// Mitsubishi GX Works2 project: plc+hmi1   PLC: Q03UDV

PROGRAM MAIN
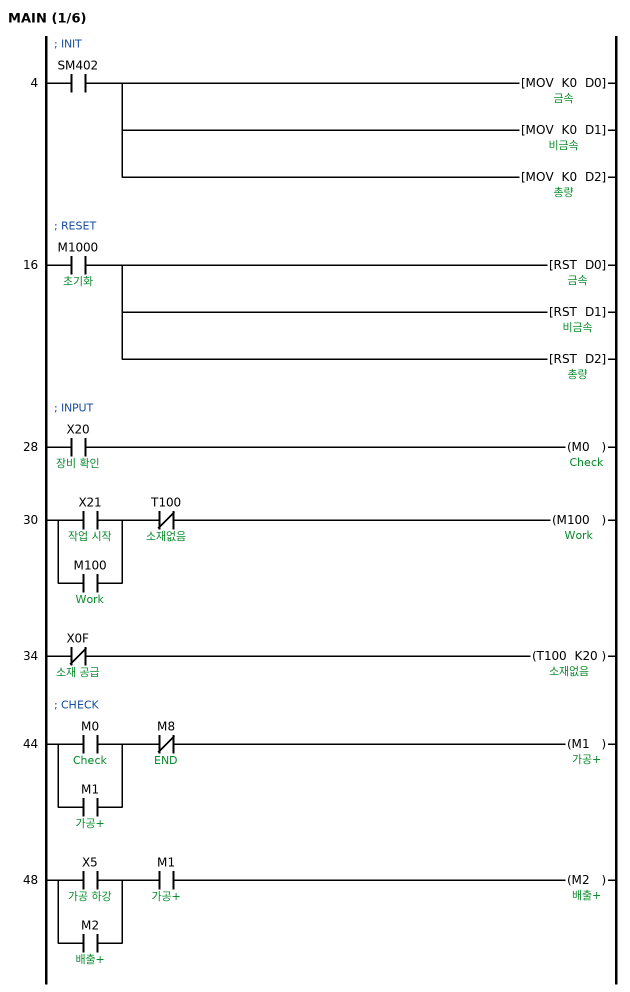
; INIT
4     LD      SM402
      MOV     K0 D0  ; 금속
      MOV     K0 D1  ; 비금속
      MOV     K0 D2  ; 총량
; RESET
16    LD      M1000  ; 초기화
      RST     D0  ; 금속
      RST     D1  ; 비금속
      RST     D2  ; 총량
; INPUT
28    LD      X20  ; 장비 확인
      OUT     M0  ; Check
30    LD      X21  ; 작업 시작
      OR      M100  ; Work
      ANI     T100  ; 소재없음
      OUT     M100  ; Work
34    LDI     X0F  ; 소재 공급
      OUT     T100 K20  ; 소재없음
; CHECK
44    LD      M0  ; Check
      OR      M1  ; 가공+
      ANI     M8  ; END
      OUT     M1  ; 가공+
48    LD      X5  ; 가공 하강
      OR      M2  ; 배출+
      AND     M1  ; 가공+
      OUT     M2  ; 배출+
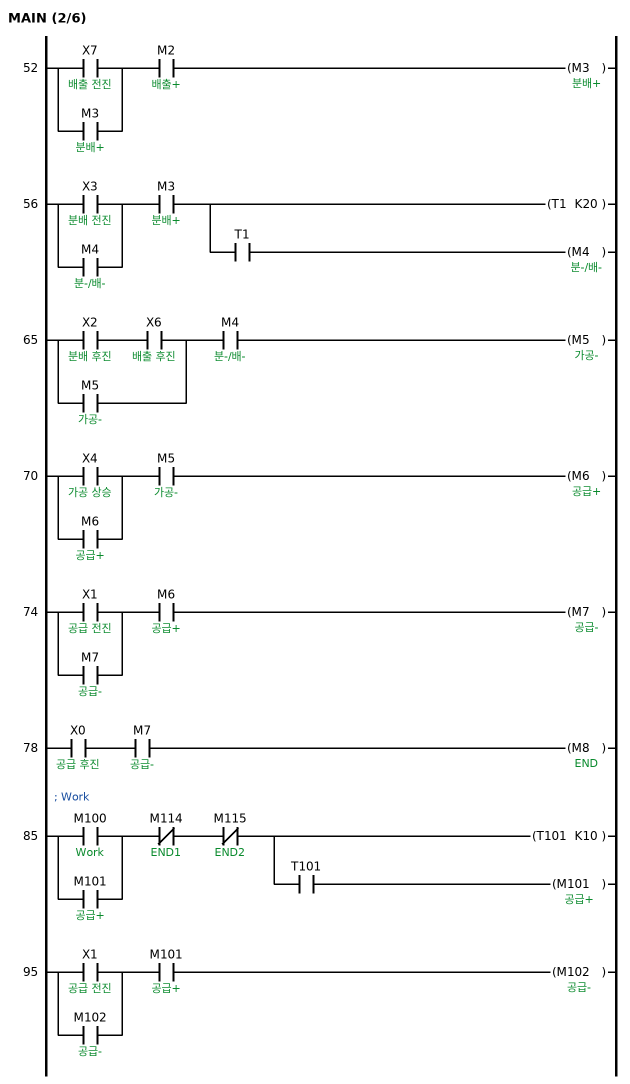
52    LD      X7  ; 배출 전진
      OR      M3  ; 분배+
      AND     M2  ; 배출+
      OUT     M3  ; 분배+
56    LD      X3  ; 분배 전진
      OR      M4  ; 분-/배-
      AND     M3  ; 분배+
      OUT     T1 K20
      AND     T1
      OUT     M4  ; 분-/배-
65    LD      X2  ; 분배 후진
      AND     X6  ; 배출 후진
      OR      M5  ; 가공-
      AND     M4  ; 분-/배-
      OUT     M5  ; 가공-
70    LD      X4  ; 가공 상승
      OR      M6  ; 공급+
      AND     M5  ; 가공-
      OUT     M6  ; 공급+
74    LD      X1  ; 공급 전진
      OR      M7  ; 공급-
      AND     M6  ; 공급+
      OUT     M7  ; 공급-
78    LD      X0  ; 공급 후진
      AND     M7  ; 공급-
      OUT     M8  ; END
; Work
85    LD      M100  ; Work
      OR      M101  ; 공급+
      ANI     M114  ; END1
      ANI     M115  ; END2
      OUT     T101 K10
      AND     T101
      OUT     M101  ; 공급+
95    LD      X1  ; 공급 전진
      OR      M102  ; 공급-
      AND     M101  ; 공급+
      OUT     M102  ; 공급-
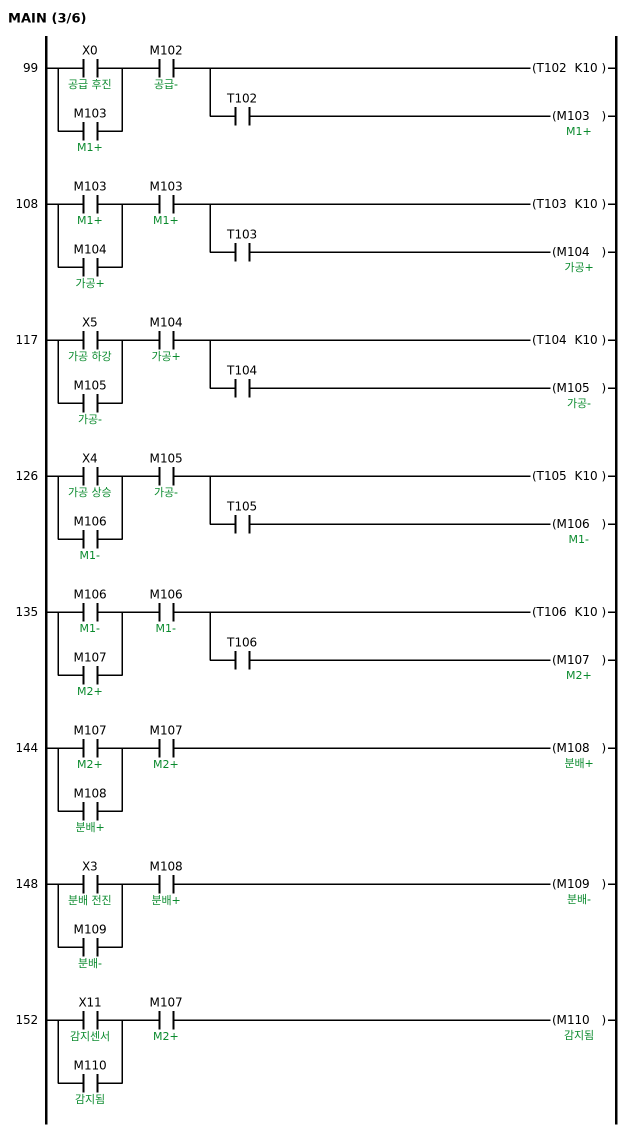
99    LD      X0  ; 공급 후진
      OR      M103  ; M1+
      AND     M102  ; 공급-
      OUT     T102 K10
      AND     T102
      OUT     M103  ; M1+
108   LD      M103  ; M1+
      OR      M104  ; 가공+
      AND     M103  ; M1+
      OUT     T103 K10
      AND     T103
      OUT     M104  ; 가공+
117   LD      X5  ; 가공 하강
      OR      M105  ; 가공-
      AND     M104  ; 가공+
      OUT     T104 K10
      AND     T104
      OUT     M105  ; 가공-
126   LD      X4  ; 가공 상승
      OR      M106  ; M1-
      AND     M105  ; 가공-
      OUT     T105 K10
      AND     T105
      OUT     M106  ; M1-
135   LD      M106  ; M1-
      OR      M107  ; M2+
      AND     M106  ; M1-
      OUT     T106 K10
      AND     T106
      OUT     M107  ; M2+
144   LD      M107  ; M2+
      OR      M108  ; 분배+
      AND     M107  ; M2+
      OUT     M108  ; 분배+
148   LD      X3  ; 분배 전진
      OR      M109  ; 분배-
      AND     M108  ; 분배+
      OUT     M109  ; 분배-
152   LD      X11  ; 감지센서
      OR      M110  ; 감지됨
      AND     M107  ; M2+
      OUT     M110  ; 감지됨
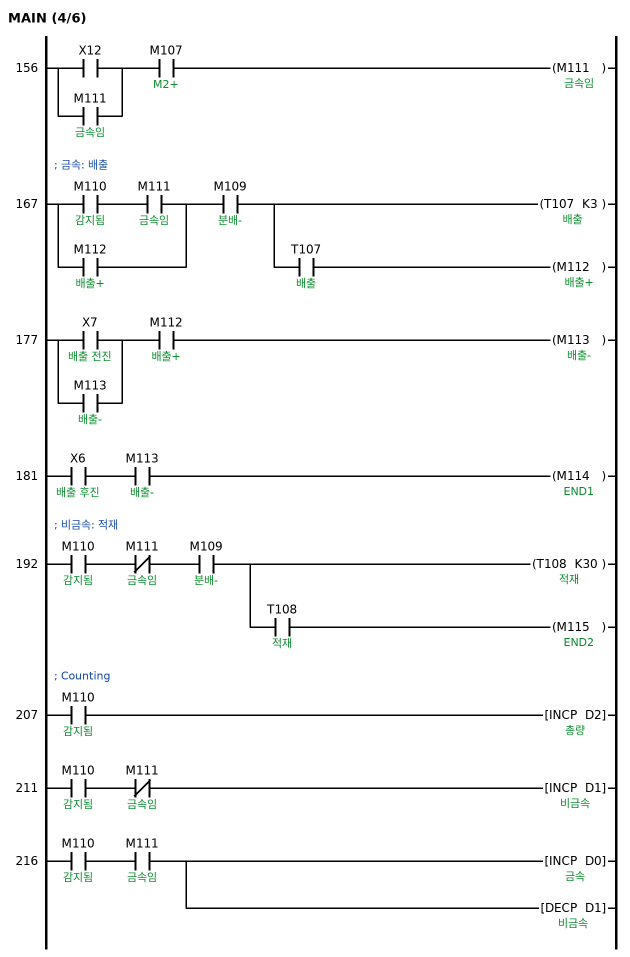
156   LD      X12
      OR      M111  ; 금속임
      AND     M107  ; M2+
      OUT     M111  ; 금속임
; 금속: 배출
167   LD      M110  ; 감지됨
      AND     M111  ; 금속임
      OR      M112  ; 배출+
      AND     M109  ; 분배-
      OUT     T107 K3  ; 배출
      AND     T107  ; 배출
      OUT     M112  ; 배출+
177   LD      X7  ; 배출 전진
      OR      M113  ; 배출-
      AND     M112  ; 배출+
      OUT     M113  ; 배출-
181   LD      X6  ; 배출 후진
      AND     M113  ; 배출-
      OUT     M114  ; END1
; 비금속: 적재
192   LD      M110  ; 감지됨
      ANI     M111  ; 금속임
      AND     M109  ; 분배-
      OUT     T108 K30  ; 적재
      AND     T108  ; 적재
      OUT     M115  ; END2
; Counting
207   LD      M110  ; 감지됨
      INCP    D2
211   LD      M110  ; 감지됨
      ANI     M111  ; 금속임
      INCP    D1
216   LD      M110  ; 감지됨
      AND     M111  ; 금속임
      INCP    D0
      DECP    D1
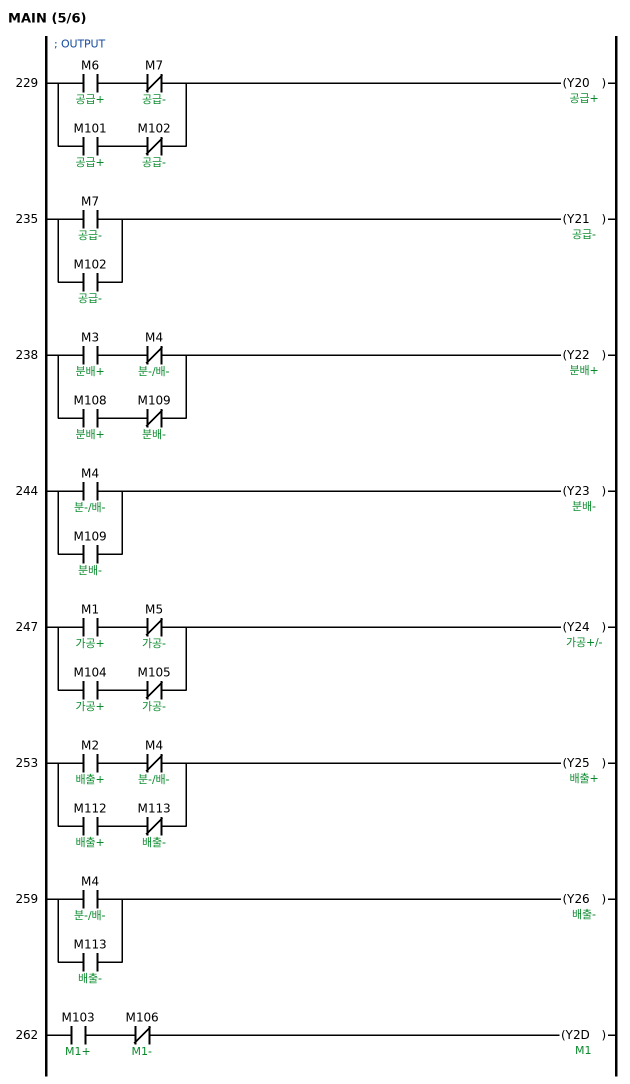
; OUTPUT
229   LD      M6  ; 공급+
      ANI     M7  ; 공급-
      LD      M101  ; 공급+
      ANI     M102  ; 공급-
      ORB
      OUT     Y20  ; 공급+
235   LD      M7  ; 공급-
      OR      M102  ; 공급-
      OUT     Y21  ; 공급-
238   LD      M3  ; 분배+
      ANI     M4  ; 분-/배-
      LD      M108  ; 분배+
      ANI     M109  ; 분배-
      ORB
      OUT     Y22  ; 분배+
244   LD      M4  ; 분-/배-
      OR      M109  ; 분배-
      OUT     Y23  ; 분배-
247   LD      M1  ; 가공+
      ANI     M5  ; 가공-
      LD      M104  ; 가공+
      ANI     M105  ; 가공-
      ORB
      OUT     Y24  ; 가공+/-
253   LD      M2  ; 배출+
      ANI     M4  ; 분-/배-
      LD      M112  ; 배출+
      ANI     M113  ; 배출-
      ORB
      OUT     Y25  ; 배출+
259   LD      M4  ; 분-/배-
      OR      M113  ; 배출-
      OUT     Y26  ; 배출-
262   LD      M103  ; M1+
      ANI     M106  ; M1-
      OUT     Y2D  ; M1
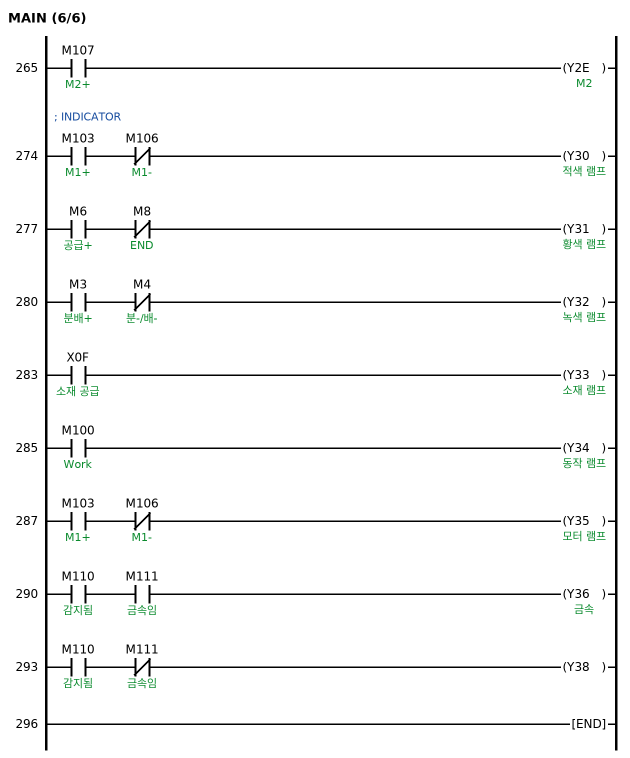
265   LD      M107  ; M2+
      OUT     Y2E  ; M2
; INDICATOR
274   LD      M103  ; M1+
      ANI     M106  ; M1-
      OUT     Y30  ; 적색 램프
277   LD      M6  ; 공급+
      ANI     M8  ; END
      OUT     Y31  ; 황색 램프
280   LD      M3  ; 분배+
      ANI     M4  ; 분-/배-
      OUT     Y32  ; 녹색 램프
283   LD      X0F  ; 소재 공급
      OUT     Y33  ; 소재 램프
285   LD      M100  ; Work
      OUT     Y34  ; 동작 램프
287   LD      M103  ; M1+
      ANI     M106  ; M1-
      OUT     Y35  ; 모터 램프
290   LD      M110  ; 감지됨
      AND     M111  ; 금속임
      OUT     Y36  ; 금속
293   LD      M110  ; 감지됨
      ANI     M111  ; 금속임
      OUT     Y38
296   END
END_PROGRAM

// device comments not shown above
M10  ; 공급 동작
M11  ; 분배 동작
M12  ; 가공 동작
M201  ; 가공+
M202  ; 가공-
M301  ; 분배+
M302  ; 분배-
